// TIA Portal V18 export
DATA_BLOCK "HMI_DB"   // DB20
// stored: AutoNumber false, InstanceOfName HMI, InstanceOfType FB
"HMI"
   // VAR
   //    DHScreen : Array[0..4] of Int;
   //    HPUScreen : Array[0..4] of Int;
   //    ConsoleScreen : Array[0..4] of Int;
   //    OscEnable : Bool := FALSE;
   //    OscAllowEn : Bool := TRUE;
   // END_VAR
   // VAR RETAIN
   //    OscBumpAdj { S7_SetPoint := 'True'} : Real := 20.0;
   // END_VAR
   // VAR
   //    OscBumpFwdInc : Bool := FALSE;
   //    OscBumpFwdDec : Bool := FALSE;
   //    OscBumpReactive : Bool := FALSE;
   //    OscBumpRevInc : Bool := FALSE;
   //    OscBumpRevDec : Bool := FALSE;
   //    OscBumpFwd : Bool := FALSE;
   //    OscBumpRev : Bool := FALSE;
   // END_VAR
   // VAR RETAIN
   //    OscBumpFwdDeg : Real := 360.0;
   //    OscBumpRevDeg : Real := 180.0;
   // END_VAR
   // VAR
   //    OscHoldButton : Bool := FALSE;
   //    OscHold : Bool := FALSE;
   //    OscBumpFwdButton : Bool;
   //    OscBumpRevButton : Bool;
   //    OscBumpFwdRevButtonEn : Bool;
   //    OscHomeRelDeg : Real := 0.0;
   // END_VAR
   // VAR RETAIN
   //    OscP1FwdMinmA { S7_SetPoint := 'True'} : Real := 250.0;
   //    OscP1FwdMaxmA { S7_SetPoint := 'True'} : Real := 700.0;
   //    OscP1RevMinmA { S7_SetPoint := 'True'} : Real := 200.0;
   //    OscP1RevMaxmA { S7_SetPoint := 'True'} : Real := 700.0;
   //    OscP1HoldmA { S7_SetPoint := 'True'} : Real := 200.0;
   //    OscP2FwdMinmA { S7_SetPoint := 'True'} : Real := 250.0;
   //    OscP2FwdMaxmA { S7_SetPoint := 'True'} : Real := 700.0;
   //    OscP2RevMinmA { S7_SetPoint := 'True'} : Real := 275.0;
   //    OscP2RevMaxmA { S7_SetPoint := 'True'} : Real := 700.0;
   //    OscP2HoldmA { S7_SetPoint := 'True'} : Real := 200.0;
   // END_VAR
   // VAR
   //    OscPosZero : Bool := FALSE;
   // END_VAR
   // VAR RETAIN
   //    OscSlewRiseFast { S7_SetPoint := 'True'} : Real := 800.0;
   //    OscSlewRiseSlow { S7_SetPoint := 'True'} : Real := 100.0;
   //    OscSlewFallFast { S7_SetPoint := 'True'} : Real := 2.5;
   //    OscSlewFallSlow { S7_SetPoint := 'True'} : Real := 2.5;
   //    OscSpeedTHper { S7_SetPoint := 'True'} : Real := 75.0;
   //    OscSpeedHoldper { S7_SetPoint := 'True'} : Real := 75.0;
   //    OscSpeedFwdRPM { S7_SetPoint := 'True'} : Real := 15.0;
   //    OscSpeedRevRPM { S7_SetPoint := 'True'} : Real := 15.0;
   // END_VAR
   // VAR
   //    OscSpeedFwdZone1 : Real := 11.25;
   //    OscSpeedFwdZone2 : Real := 12.75;
   //    OscSpeedFwdZone3 : Real := 11.25;
   //    OscSpeedFwdZone4 : Real := 12.0;
   //    OscSpeedRevZone1 : Real := 11.25;
   //    OscSpeedRevZone2 : Real := 12.75;
   //    OscSpeedRevZone3 : Real := 11.25;
   //    OscSpeedRevZone4 : Real := 12.0;
   //    OscStart : Bool := FALSE;
   //    OscStartButton : Bool := FALSE;
   //    OscStop : Bool := FALSE;
   //    OscStopButton : Bool := TRUE;
   // END_VAR
   // VAR RETAIN
   //    OscTorqAdj { S7_SetPoint := 'True'} : Real := 500.0;
   //    OscTorqFwdFtLbs : Real := 10000.0;
   // END_VAR
   // VAR
   //    OscTorqFwdInc : Bool := FALSE;
   //    OscTorqFwdDec : Bool := FALSE;
   //    OscTorqRevInc : Bool := FALSE;
   // END_VAR
   // VAR RETAIN
   //    OscTorqRevFtLbs : Real := 10000.0;
   // END_VAR
   // VAR
   //    OscTorqRevDec : Bool := FALSE;
   //    OscTorqSetPSI : Real := 1725.63;
   // END_VAR
   // VAR RETAIN
   //    OscTurnAdj { S7_SetPoint := 'True'} : Real := 0.25;
   //    OscTurnFwd : Real := 2.0;
   // END_VAR
   // VAR
   //    OscTurnFwdInc : Bool := FALSE;
   //    OscTurnFwdDec : Bool := FALSE;
   // END_VAR
   // VAR RETAIN
   //    OscTurnRev : Real := 2.0;
   // END_VAR
   // VAR
   //    OscTurnRevInc : Bool := FALSE;
   //    OscTurnRevDec : Bool := FALSE;
   //    OscTorqFwdLowLimFtlbs : Real := 9000.0;
   //    OscTorqFwdHighLimFtLbs : Real := 9700.0;
   //    OscTorqRevLowLimFtlbs : Real := 9000.0;
   //    OscTorqRevHighLimFtLbs : Real := 9700.0;
   //    OscHomeLowRelDeg : Real := -376.3636;
   //    OscHomeLow2RelDeg : Real := -752.7273;
   //    OscHomeHighRelDeg : Real := 16.36364;
   //    OscHomeHigh2RelDeg : Real := 32.72727;
   //    OscPosDeg : Real := -1227.273;
   //    SpareVolts : Real := 0.0;
   //    Spare4MA : Real := 4.0;
   //    LampTest : Bool := FALSE;
   //    LampTestLamp_TP { S7_SetPoint := 'True'} : TP_TIME;
   //    LampTestHorn_TP { S7_SetPoint := 'True'} : TP_TIME;
   //    ScreenNameInvis { S7_SetPoint := 'True'} : Bool := FALSE;
   //    ScreenBypassVis : Bool := FALSE;
   //    ScreenLampTestVis : Bool := FALSE;
   //    HornSilence_TOF { S7_SetPoint := 'True'} : TOF_TIME;
   //    HornSilenceReset { S7_SetPoint := 'True'} : Bool := FALSE;
   //    Alarms1 : Int := 0;
   //    Alarms2 : Int := 7104;
   //    Warnings1 : Int := 1;
   //    Alarms1_To_Unified : Array[0..15] of Bool;
   //    Alarms2_To_Unified : Array[0..15] of Bool;
   //    Warnings1_To_Unified : Array[0..15] of Bool;
   // END_VAR
BEGIN
   DHScreen[0..4] := 0;
   HPUScreen[0..1] := 1;
   HPUScreen[2] := 0;
   HPUScreen[3] := 1;
   HPUScreen[4] := 0;
   ConsoleScreen[0..1] := 1;
   ConsoleScreen[2] := 0;
   ConsoleScreen[3] := 1;
   ConsoleScreen[4] := 0;
   LampTestLamp_TP.PT := T#0MS;
   LampTestLamp_TP.IN := FALSE;
   LampTestHorn_TP.PT := T#0MS;
   LampTestHorn_TP.IN := FALSE;
   HornSilence_TOF.PT := T#0MS;
   HornSilence_TOF.IN := FALSE;
   Alarms1_To_Unified[0..15] := FALSE;
   Alarms2_To_Unified[0..5] := FALSE;
   Alarms2_To_Unified[6..9] := TRUE;
   Alarms2_To_Unified[10] := FALSE;
   Alarms2_To_Unified[11..12] := TRUE;
   Alarms2_To_Unified[13..15] := FALSE;
   Warnings1_To_Unified[0] := TRUE;
   Warnings1_To_Unified[1..15] := FALSE;
END_DATA_BLOCK
